// Generic analog input conditioner.
//
// Pipeline:
//   UNION terminal -> type select -> quality gate -> clamp to scaling range
//   -> linear EU scaling -> optional first-order LPF -> sts
//
// The UNION input (inRaw) means one FB instance handles any raw form the
// hardware produces â€” 0-10 V (INT), 4-20 mA (INT), 32-bit counter (UDINT),
// scaled REAL, bit-packed WORD, etc. Pick the interpretation with
// cfg.inputType.
//
// Scope: conditioning only. Process-alarm limits (HH / HI / LO / LL),
// latching, severity, and ack all live on FB_AlarmLimit â€” compose it with
// sts.value if you need that behaviour. Faults here are restricted to
// ground truths about the signal itself (quality, clamp, bad config).
{attribute 'OPC.UA.DA' := '1'}
FUNCTION_BLOCK FB_AnalogInput EXTENDS FB_DeviceBase
VAR_INPUT
    {attribute 'OPC.UA.DA' := '0'}
    inRaw : U_IoRaw_In;
    {attribute 'OPC.UA.DA' := '1'}
    {attribute 'OPC.UA.DA.Access' := '1'}
    cfg        : ST_AnalogInput_Cfg;
    {attribute 'OPC.UA.DA' := '0'}
    inpQuality : E_IO_Quality := E_IO_Quality.GOOD;
END_VAR

VAR_OUTPUT
    {attribute 'OPC.UA.DA' := '1'}
    {attribute 'OPC.UA.DA.Access' := '1'}
    sts : ST_AnalogInput_Sts;
END_VAR

VAR
    _inputSnapshot : U_IoRaw_In;
    _lastConditioningCfg : ST_AnalogInput_Cfg;
    _conditioningCfgKnown : BOOL;
    _hasValidSample : BOOL;
    _reseedPending : BOOL;

    // Commissioning state.
    {attribute 'OPC.UA.DA' := '0'}
    _firstScan     : BOOL := TRUE;
    {attribute 'OPC.UA.DA' := '0'}
    _configBad     : BOOL;
    {attribute 'OPC.UA.DA' := '0'}
    _taskDtSec     : REAL;

    // Filter + watchdog timers.
    {attribute 'OPC.UA.DA' := '0'}
    _filter        : FB_LPF_FirstOrder_IIR;
    {attribute 'OPC.UA.DA' := '0'}
    _tonBadQuality : TON;

    // Scratch values (reset every scan).
    {attribute 'OPC.UA.DA' := '0'}
    _rawReal       : REAL;
    _scaledWide    : LREAL;
    _signalBad     : BOOL;
    {attribute 'OPC.UA.DA' := '0'}
    _clampedRaw    : REAL;
    {attribute 'OPC.UA.DA' := '0'}
    _scaledReal    : REAL;
    {attribute 'OPC.UA.DA' := '0'}
    _finalReal     : REAL;
END_VAR

_ProcessOperatorCommands();
// 1. First scan: config validation + task dt cache for the filter.
IF _firstScan THEN
    _firstScan := FALSE;
    _taskDtSec := TIME_TO_REAL(F_GetTaskCycleTime()) / 1000.0;

END_IF;

// Classify representations before comparisons; NaN comparisons can stop the PLC.
_configBad := NOT F_IsFiniteReal(value := cfg.euMin) OR NOT F_IsFiniteReal(value := cfg.euMax) OR
              NOT F_IsFiniteReal(value := cfg.rawMin) OR NOT F_IsFiniteReal(value := cfg.rawMax);
IF NOT _configBad THEN
    _configBad := NOT cfg.useRawValue AND (cfg.rawMin >= cfg.rawMax OR cfg.euMin >= cfg.euMax);
END_IF;
_configBad := _configBad OR NOT (
    cfg.inputType = __SYSTEM.TYPE_CLASS.TYPE_INT OR cfg.inputType = __SYSTEM.TYPE_CLASS.TYPE_UINT OR
    cfg.inputType = __SYSTEM.TYPE_CLASS.TYPE_WORD OR cfg.inputType = __SYSTEM.TYPE_CLASS.TYPE_DINT OR
    cfg.inputType = __SYSTEM.TYPE_CLASS.TYPE_UDINT OR cfg.inputType = __SYSTEM.TYPE_CLASS.TYPE_DWORD OR
    cfg.inputType = __SYSTEM.TYPE_CLASS.TYPE_REAL);

// Only compare validated configurations; previous snapshots contain finite values.
IF NOT _configBad THEN
    IF _conditioningCfgKnown AND _hasValidSample THEN
        IF cfg.inputType <> _lastConditioningCfg.inputType OR
           cfg.useRawValue <> _lastConditioningCfg.useRawValue OR
           cfg.rawMin <> _lastConditioningCfg.rawMin OR cfg.rawMax <> _lastConditioningCfg.rawMax OR
           cfg.euMin <> _lastConditioningCfg.euMin OR cfg.euMax <> _lastConditioningCfg.euMax OR
           ((cfg.filterTau = T#0MS) <> (_lastConditioningCfg.filterTau = T#0MS)) THEN
            _reseedPending := TRUE;
        END_IF;
    END_IF;
    _lastConditioningCfg := cfg;
    _conditioningCfgKnown := TRUE;
END_IF;

sts.unit    := cfg.unit;
sts.quality := inpQuality;

// 2. Snapshot the selected source.
_inputSnapshot := inRaw;
CASE cfg.inputType OF
    __SYSTEM.TYPE_CLASS.TYPE_INT:   _rawReal := TO_REAL(_inputSnapshot.nInt);
    __SYSTEM.TYPE_CLASS.TYPE_UINT:  _rawReal := TO_REAL(_inputSnapshot.ui);
    __SYSTEM.TYPE_CLASS.TYPE_WORD:  _rawReal := TO_REAL(_inputSnapshot.w);
    __SYSTEM.TYPE_CLASS.TYPE_DINT:  _rawReal := TO_REAL(_inputSnapshot.di);
    __SYSTEM.TYPE_CLASS.TYPE_UDINT: _rawReal := TO_REAL(_inputSnapshot.udi);
    __SYSTEM.TYPE_CLASS.TYPE_DWORD: _rawReal := TO_REAL(_inputSnapshot.dw);
    __SYSTEM.TYPE_CLASS.TYPE_REAL:
    _rawReal := _inputSnapshot.fReal;
ELSE
    _rawReal := sts.rawReal;
END_CASE;

// 3. Quality-gated hold. Ignore the freshly read value while BAD.
_signalBad := NOT F_IsFiniteReal(value := _rawReal);
IF _signalBad OR _configBad THEN sts.quality := E_IO_Quality.BAD; END_IF;
IF _signalBad OR _configBad OR NOT (inpQuality = E_IO_Quality.GOOD OR inpQuality = E_IO_Quality.CLAMPED) THEN
    _rawReal := sts.rawReal;
END_IF;

sts.rawReal := _rawReal;

// Unusable samples cannot advance conditioning state or reinterpret held raw data.
// Preserve the last published value and filter history until a valid sample arrives.
_finalReal := sts.value;
IF NOT _configBad AND NOT _signalBad AND
   (inpQuality = E_IO_Quality.GOOD OR inpQuality = E_IO_Quality.CLAMPED) THEN
// 4. Raw-value bypass â€” no clamp / scale / filter.
IF cfg.useRawValue THEN
    _finalReal         := _rawReal;
    sts.scaled      := _rawReal;
    sts.clampedLow  := FALSE;
    sts.clampedHigh := FALSE;
    sts.clampActive := FALSE;
ELSE
    // 4a. Clamp-and-report against the scaling range. The same comparison
    //     drives both the scaling clamp and the sts.clamped* booleans so the
    //     HMI surface always matches what the math actually used.
    sts.clampedLow  := _rawReal < cfg.rawMin;
    sts.clampedHigh := _rawReal > cfg.rawMax;
    sts.clampActive := sts.clampedLow OR sts.clampedHigh;

    _clampedRaw := _rawReal;
    IF sts.clampedLow THEN
        _clampedRaw := cfg.rawMin;
    ELSIF sts.clampedHigh THEN
        _clampedRaw := cfg.rawMax;
    END_IF;

    // Promote quality tag while clamped (even if no fault is raised).
    IF sts.clampActive AND sts.quality = E_IO_Quality.GOOD THEN
        sts.quality := E_IO_Quality.CLAMPED;
    END_IF;

    // Wide intermediate math avoids overflow before range checks can act.
    IF NOT _configBad THEN
        _scaledWide := REAL_TO_LREAL(cfg.euMin)
            + (REAL_TO_LREAL(_clampedRaw) - REAL_TO_LREAL(cfg.rawMin))
            * (REAL_TO_LREAL(cfg.euMax) - REAL_TO_LREAL(cfg.euMin))
            / (REAL_TO_LREAL(cfg.rawMax) - REAL_TO_LREAL(cfg.rawMin));
        _scaledReal := LREAL_TO_REAL(LIMIT(LREAL#-3.402823E38, _scaledWide, LREAL#3.402823E38));
    ELSE
        _scaledReal := sts.value;
        sts.quality := E_IO_Quality.BAD;
    END_IF;
    sts.scaled := _scaledReal;

    // 4c. Optional first-order LPF. Pass-through when tau is 0.
    IF cfg.filterTau <> T#0MS THEN
        IF _reseedPending THEN
            _filter.Seed(value := REAL_TO_LREAL(_scaledReal));
        END_IF;
        _filter(
            fInput := _scaledReal,
            fDt    := _taskDtSec,
            fTau   := TIME_TO_REAL(cfg.filterTau) / 1000.0
        );
        _finalReal := LREAL_TO_REAL(_filter.fOutput);
    ELSE
        _finalReal := _scaledReal;
    END_IF;
END_IF;
_hasValidSample := TRUE;
_reseedPending := FALSE;
ELSE
    sts.clampedLow := FALSE;
    sts.clampedHigh := FALSE;
    sts.clampActive := FALSE;
END_IF;

sts.value := _finalReal;

// 5. Quality watchdog.
_tonBadQuality(
    IN := (_signalBad OR NOT (inpQuality = E_IO_Quality.GOOD OR inpQuality = E_IO_Quality.CLAMPED)) AND cfg.qualityFaultAfter > T#0MS,
    PT := cfg.qualityFaultAfter
);

// 6. Single-source-of-truth fault raise. See _RaiseActiveFault for priority.
_RaiseActiveFault();

// 7. Refresh shared header.
_UpdateHeader(header := sts.header, stateString := '', busy := FALSE);

// Pick the highest-severity active fault and raise it. Priority:
//   BadConfig (commissioning)
//   BadQuality (watchdog)
//   ClampHigh / ClampLow (if clampAsFault)
//
// If no rule applies the active fault (if any) is cleared so the device
// auto-recovers when the condition goes away.
METHOD PROTECTED _RaiseActiveFault
VAR
    code   : DINT;
    source : STRING(31);
    reason : STRING(79);
END_VAR
code := 0;

IF _configBad THEN
    code   := E_AnalogInput_Fault.BadConfig;
    source := 'CONFIG';
    reason := 'rawMin >= rawMax or euMin > euMax';
ELSIF _tonBadQuality.Q THEN
    code   := E_AnalogInput_Fault.BadQuality;
    source := 'QUALITY';
    reason := 'inpQuality stayed BAD past qualityFaultAfter';
ELSIF cfg.clampAsFault AND sts.clampedHigh THEN
    code   := E_AnalogInput_Fault.ClampHigh;
    source := 'CLAMP_H';
    reason := CONCAT('Raw reading above RawMax=', REAL_TO_STRING(cfg.rawMax));
ELSIF cfg.clampAsFault AND sts.clampedLow THEN
    code   := E_AnalogInput_Fault.ClampLow;
    source := 'CLAMP_L';
    reason := CONCAT('Raw reading below RawMin=', REAL_TO_STRING(cfg.rawMin));
END_IF;

IF code = 0 THEN
    IF IsFaulted() THEN
        _ClearFault();
    END_IF;
ELSE
    _Raise(
        code   := code,
        source := source,
        reason := reason
    );
END_IF;
END_METHOD

METHOD PROTECTED ResolveFaultString : STRING(79)
VAR_INPUT
    code : DINT;
END_VAR
CASE code OF
    0:
        ResolveFaultString := '';
    E_AnalogInput_Fault.BadQuality:
        ResolveFaultString := 'Signal quality BAD past configured timeout';
    E_AnalogInput_Fault.ClampLow:
        ResolveFaultString := 'Raw reading below RawMin';
    E_AnalogInput_Fault.ClampHigh:
        ResolveFaultString := 'Raw reading above RawMax';
    E_AnalogInput_Fault.BadConfig:
        ResolveFaultString := 'Invalid scaling range configured';
ELSE
    ResolveFaultString := CONCAT('AnalogInput fault ', DINT_TO_STRING(code));
END_CASE;
END_METHOD

// Owning-task application API: invalidate history when binding a different source.
// Call before supplying its first fresh sample; this is not a remote command.
METHOD PUBLIC ReassignInput
_hasValidSample := FALSE;
_reseedPending := TRUE;
sts.value := 0.0;
sts.scaled := 0.0;
sts.rawReal := 0.0;
sts.quality := E_IO_Quality.UNKNOWN;
sts.clampedLow := FALSE;
sts.clampedHigh := FALSE;
sts.clampActive := FALSE;
_tonBadQuality(IN := FALSE);
END_METHOD

END_FUNCTION_BLOCK

(* stored: Version 1.1.0.1, ProductVersion 3.1.4026.12
   POU FB_AnalogInput: Id {a0100003-0000-0000-0000-000000000001}, SpecialFunc None
   Folder Configuration: Id {8a55965b-c382-56bd-bd8b-a40c6f65522e}
   Folder Protected: Id {a0100003-0000-0000-f000-000000000001}
   Method _RaiseActiveFault: Id {a0100003-0000-0000-1000-000000000001}
   Method ResolveFaultString: Id {a0100003-0000-0000-1000-000000000002}
   Method ReassignInput: Id {6556c42d-9c68-4e18-b0bd-a1246f50908a} *)
